TYPE ST_PROCESS :
STRUCT
	ChageSlot:			BOOL:=FALSE;	(* Change slot after finished this position TASK *)	
	ProcessType:		ENUM_PROCESS;		(* Describe what we want to do in *)
	Comment:			STRING(255);
	Parameter:			STRING(255);
END_STRUCT
END_TYPE

(* stored: Version 1.1.0.1, ProductVersion 3.1.4024.10
   DUT ST_PROCESS: Id {0ed5c5cf-870c-4583-8e34-6fb395961947} *)
